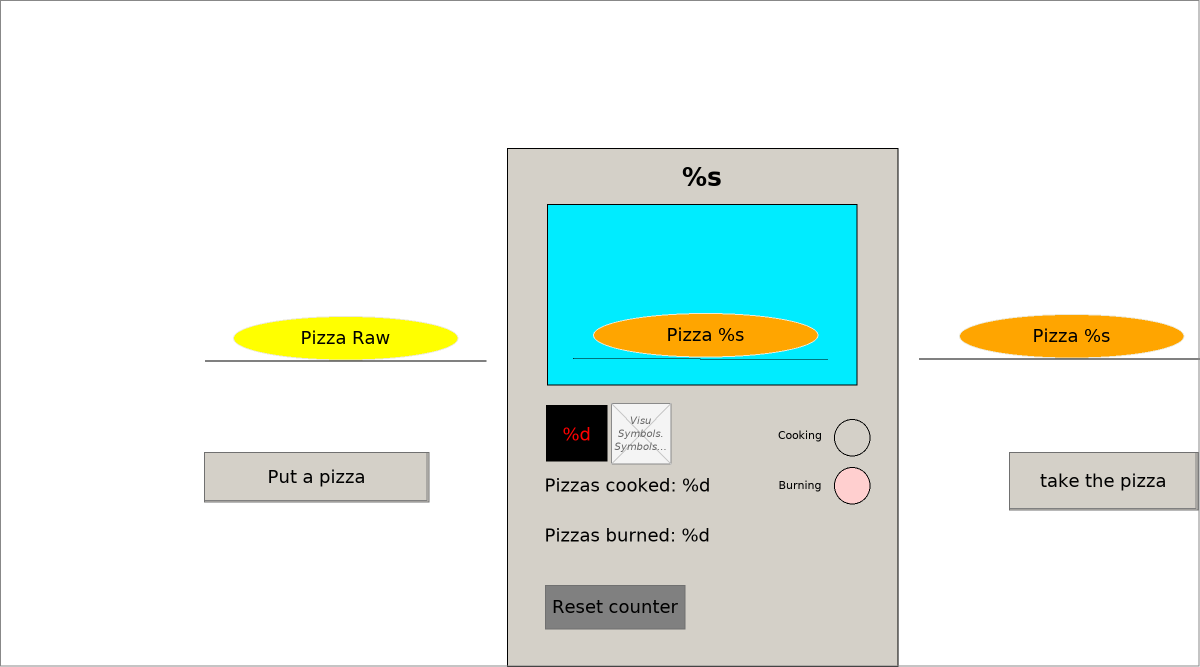
VISUALIZATION OvenSimulation  // 1200x667
    Rectangle (507,148 391x519)
    Ellipse (233,316 225x44), "Pizza Raw", invisible if: NOT main.fbMyPizzaOven.bs_PizzaOnEntrit
    Rectangle (546,405 61x56)
    Rectangle (547,204 310x181)
    Line (573,358) (827,359)
    Line (1200,359) (919,359)
    Line (486,361) (205,361)
    Ellipse (593,313 225x44), "Pizza %s", text variable: MAIN.fbMyPizzaOven.sPizzaDescription, colour toggle: MAIN.fbMyPizzaOven.bBurnt, invisible if: NOT main.fbMyPizzaOven.bs_PizzaOnOven
    Ellipse (834,419 36x37), colour toggle: MAIN.fbMyPizzaOven.LightCooking
    Ellipse (834,467 36x37), colour toggle: MAIN.fbMyPizzaOven.LBuzzer
    Label (744,403 112x65), "Cooking"
    Label (744,453 112x65), "Burning"
    Rectangle (497,413 160x43), "%d", text variable: MAIN.fbMyPizzaOven.sCookingTime, invisible if: not MAIN.fbMyPizzaOven.LightCooking
    Rectangle (507,153 390x47), "%s", text variable: MAIN.fbMyPizzaOven.sStateDescription
    Rectangle (516,462 223x47), "Pizzas cooked: %d", text variable: MAIN.fbMyPizzaOven.iTotalPizzasCooked
    Button (204,452 225x50), "Put a pizza"
        OnMouseDown: execute { main.btn_PutAPizza:=TRUE; }
        OnMouseUp: execute { main.btn_PutAPizza:=FALSE; }
    Button (1009,452 189x58), "take the pizza"
        OnMouseDown: execute { main.btn_PackageThePizza:=TRUE; }
        OnMouseUp: execute { main.btn_PackageThePizza:=FALSE; }
    Button (545,585 140x44), "Reset counter"
        OnMouseDown: execute { main.bReset:=TRUE; }
        OnMouseUp: execute { main.bReset:=FALSE; }
    Ellipse (959,314 225x44), "Pizza %s", text variable: MAIN.fbMyPizzaOven.sPizzaDescription2, colour toggle: MAIN.fbMyPizzaOven.bBurnt2, invisible if: NOT main.fbMyPizzaOven.bs_PizzaOnExit
    Rectangle (516,512 223x47), "Pizzas burned: %d", text variable: MAIN.fbMyPizzaOven.iTotalPizzasBurned
    Image (611,403 60x61), image: VisuSymbols.Symbols.Timer
END_VISUALIZATION

(* stored: Version 1.1.0.1, ProductVersion 3.1.4024.3
   Visu OvenSimulation: Id {cf67f018-acde-4636-b51a-9996667c6a6d} *)
